Staubli VAL3: getFrameId.pgx

public program getFrameId(num& x_nFrame)
begin
  // give back the frame
  x_nFrame=jEditPoint.nIndexFrame
end
